FUNCTION_BLOCK Test_ReadWriteBySymbolName EXTENDS T_UnitTestBase
VAR
    AdsPort                  : UINT;
    AdsReadWriteBySymbolName : T_AdsReadWriteBySymbolName;
    AdsReadSymbolName        : T_AdsReadSymbolName;
    TestInteger              : T_Integer;
    State                    : INT;
END_VAR

METHOD Init
State := 0;
END_METHOD

{attribute 'analysis' := '-33'} // inhibit unused variable warning
METHOD RunTest
VAR_OUTPUT
    TestCompleted : BOOL;
    TestFailed    : BOOL;
END_VAR
VAR_INST
    SymbolName      : T_MaxString;
    ReadWriteResult : INT;
END_VAR
CASE State OF
    0:
        AdsPort := _AppInfo.AdsPort;
        TestInteger.Init(1111);
        ReadWriteResult := 0;
        AdsReadSymbolName.Execute(Address := ADR(TestInteger),
                                  Length  := SIZEOF(TestInteger),
                                  PlcPort := AdsPort);
        State := 10;

    10:
        IF NOT AdsReadSymbolName.Execution.Busy THEN
            SymbolName := CONCAT(AdsReadSymbolName.SymbolName, '#Inc');
            State      := 20;
        END_IF

    20:
        AdsReadWriteBySymbolName.Execute(AmsNetId         := '',
                                         Port             := AdsPort,
                                         SymbolName       := SymbolName,
                                         ReadDataAddress  := ADR(ReadWriteResult),
                                         ReadDataLength   := SIZEOF(ReadWriteResult),
                                         WriteDataAddress := 0,
                                         WriteDataLength  := 0,
                                         KeepSymbolHandle := FALSE);

        State := 30;

    30:
        IF NOT AdsReadWriteBySymbolName.Execution.Busy THEN
            State := 40;
        END_IF

    40:
        AssertTrue(Source    := TestName,
                   Condition := (ReadWriteResult = 1112),
                   Message   := 'ReadWriteResult <> 1112',
                   Failed    => TestFailed);

        TestCompleted := TRUE;
END_CASE

AdsReadWriteBySymbolName();
AdsReadSymbolName();
END_METHOD

END_FUNCTION_BLOCK

(* stored: Version 1.1.0.1, ProductVersion 3.1.4024.12
   POU Test_ReadWriteBySymbolName: Id {957952f4-750d-06be-083a-2dd0a58feaab}, SpecialFunc None
   Method Init: Id {927c5017-e915-058e-379e-68311b9ee171}
   Method RunTest: Id {74234455-1e06-043d-04c5-26fb7056d87a} *)
